FUNCTION BundleIsValid : BOOL
VAR_INPUT
	b : REFERENCE TO Bundle;
END_VAR

BundleIsValid := NOT(b.id = '');

END_FUNCTION

(* stored: Version 1.1.0.1, ProductVersion 3.1.4024.11
   POU BundleIsValid: Id {10192e08-9c9e-4199-98a2-e54aea68a69b}, SpecialFunc None *)
